// TIA Portal V19 export
FUNCTION "InputMinne" : Void   // FC1, LAD
{ S7_Optimized_Access := 'TRUE' }
// stored: SetENOAutomatically false
BEGIN

REGION Network 1
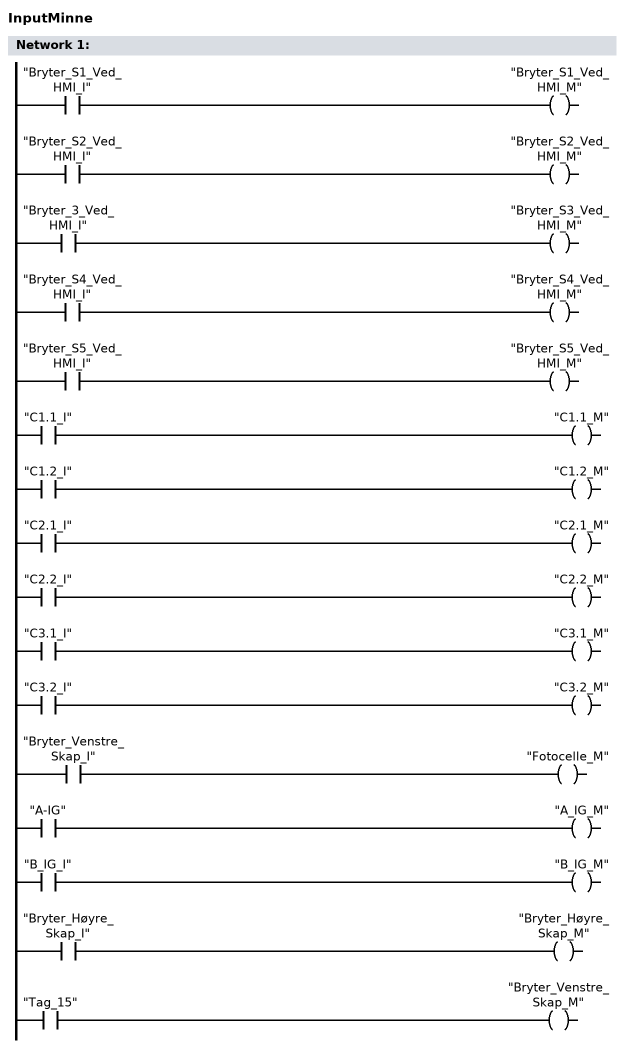
   RUNG wire#powerrail
      Contact( "Bryter_S1_Ved_HMI_I" )
      Coil( "Bryter_S1_Ved_HMI_M" )
   END_RUNG
   RUNG wire#powerrail
      Contact( "Bryter_S2_Ved_HMI_I" )
      Coil( "Bryter_S2_Ved_HMI_M" )
   END_RUNG
   RUNG wire#powerrail
      Contact( "Bryter_3_Ved_HMI_I" )
      Coil( "Bryter_S3_Ved_HMI_M" )
   END_RUNG
   RUNG wire#powerrail
      Contact( "Bryter_S4_Ved_HMI_I" )
      Coil( "Bryter_S4_Ved_HMI_M" )
   END_RUNG
   RUNG wire#powerrail
      Contact( "Bryter_S5_Ved_HMI_I" )
      Coil( "Bryter_S5_Ved_HMI_M" )
   END_RUNG
   RUNG wire#powerrail
      Contact( "C1.1_I" )
      Coil( "C1.1_M" )
   END_RUNG
   RUNG wire#powerrail
      Contact( "C1.2_I" )
      Coil( "C1.2_M" )
   END_RUNG
   RUNG wire#powerrail
      Contact( "C2.1_I" )
      Coil( "C2.1_M" )
   END_RUNG
   RUNG wire#powerrail
      Contact( "C2.2_I" )
      Coil( "C2.2_M" )
   END_RUNG
   RUNG wire#powerrail
      Contact( "C3.1_I" )
      Coil( "C3.1_M" )
   END_RUNG
   RUNG wire#powerrail
      Contact( "C3.2_I" )
      Coil( "C3.2_M" )
   END_RUNG
   RUNG wire#powerrail
      Contact( "Bryter_Venstre_Skap_I" )
      Coil( "Fotocelle_M" )
   END_RUNG
   RUNG wire#powerrail
      Contact( "A-IG" )
      Coil( "A_IG_M" )
   END_RUNG
   RUNG wire#powerrail
      Contact( "B_IG_I" )
      Coil( "B_IG_M" )
   END_RUNG
   RUNG wire#powerrail
      Contact( "Bryter_Høyre_Skap_I" )
      Coil( "Bryter_Høyre_Skap_M" )
   END_RUNG
   RUNG wire#powerrail
      Contact( "Tag_15" )
      Coil( "Bryter_Venstre_Skap_M" )
   END_RUNG
   // the same network as SCL:
   "Bryter_S1_Ved_HMI_M" := "Bryter_S1_Ved_HMI_I";
   "Bryter_S2_Ved_HMI_M" := "Bryter_S2_Ved_HMI_I";
   "Bryter_S3_Ved_HMI_M" := "Bryter_3_Ved_HMI_I";
   "Bryter_S4_Ved_HMI_M" := "Bryter_S4_Ved_HMI_I";
   "Bryter_S5_Ved_HMI_M" := "Bryter_S5_Ved_HMI_I";
   "C1.1_M" := "C1.1_I";
   "C1.2_M" := "C1.2_I";
   "C2.1_M" := "C2.1_I";
   "C2.2_M" := "C2.2_I";
   "C3.1_M" := "C3.1_I";
   "C3.2_M" := "C3.2_I";
   "Fotocelle_M" := "Bryter_Venstre_Skap_I";
   "A_IG_M" := "A-IG";
   "B_IG_M" := "B_IG_I";
   "Bryter_Høyre_Skap_M" := "Bryter_Høyre_Skap_I";
   "Bryter_Venstre_Skap_M" := "Tag_15";
END_REGION
END_FUNCTION
